FUNCTION_BLOCK Zona2 EXTENDS ZONA
VAR_INPUT	

Enable	:	BOOL;
EMG		:	BOOL;
Ripristino : BOOL;
a_0 : BOOL;
a_1	: BOOL;
I5 : BOOL;
Trigger_I : BOOL;
libero_I  : BOOL;
END_VAR
VAR_OUTPUT
	
Q1 : BOOL;
Q2 : BOOL;
Trigger_O : BOOL;
libero_O : BOOL;
END_VAR

VAR	
stato : (S_attesa, S_uscita, S_Rientro, S_Ripristino, S_Emergenza) := S_attesa;
S_attesa : BOOL;
S_Uscita : BOOL;
S_rientro : BOOL;
S_ripristino : BOOL;
S_emergenza  : BOOL;

END_VAR

//Comandi transizione degli stati

IF EMG = FALSE  OR Enable = FALSE THEN
	
	stato := S_Emergenza
	
END_IF

CASE stato OF
	S_Emergenza:
	
		IF Enable = TRUE AND Ripristino = TRUE THEN
		
			stato := S_Ripristino;
		
		END_IF
		
		Q1 := FALSE;
		Q2 := FALSE;
		Libero_O := FALSE;
		
	S_Ripristino:
		
		IF Enable = TRUE AND a_0 = TRUE THEN
			
			stato := S_Attesa;
			
		END_IF
	
	S_Attesa: 
	
		IF Enable = TRUE AND Trigger_I = TRUE AND Libero_I = TRUE AND a_0 = TRUE THEN
			
			stato := S_Uscita;
			
		END_IF
	
		Q1 := FALSE;
		Q2 := FALSE;
		Libero_O := TRUE;
	
	S_Uscita:
	
		IF a_1 = TRUE THEN
			
			stato := S_Rientro;
			
		END_IF
	
		Q1 := FALSE;
		Q2 := TRUE;
		Libero_O := FALSE;
	
	S_Rientro:
	
		IF a_0 = TRUE THEN
			
			stato := S_Attesa;
			
		END_IF
	
		Q1 := TRUE;
		Q2 := FALSE;
		Libero_O := FALSE;

END_CASE

END_FUNCTION_BLOCK

(* stored: Version 1.1.0.1, ProductVersion 3.1.4024.12
   POU Zona2: Id {6dde8437-606b-4d0e-8b96-5f698fbf635a}, SpecialFunc None *)
